TYPE ST_StationStatus EXTENDS ST_Status :
STRUCT
	eState	: E_StationState;
	sName	: STRING(31);
END_STRUCT
END_TYPE

(* stored: Version 1.1.0.1, ProductVersion 3.1.4024.12
   DUT ST_StationStatus: Id {0183bd08-1fa6-485a-92b8-01229c97de83} *)
